FUNCTION_BLOCK FB_FieldCodecEnum EXTENDS FB_FieldCodec
VAR_INPUT
END_VAR
VAR_OUTPUT
END_VAR
VAR
	nValue : DINT;
END_VAR

METHOD CalculatePackedDataSize : HRESULT
VAR_INPUT CONSTANT
	anyFirstElem	: T_Any;
	nLength	        : UDINT;        // items to write
END_VAR
VAR_OUTPUT
    nPackedDataSize : UDINT;
END_VAR
VAR
    anyItem         : T_ANY;
    i               : UDINT;
END_VAR
IF anyFirstElem.pValue = NULL OR anyFirstElem.TypeClass <> __SYSTEM.TYPE_CLASS.TYPE_ENUM THEN
    CalculatePackedDataSize := E_HRESULTAdsErr.INVALIDDATA;
    RETURN;
END_IF

anyItem := anyFirstElem;

IF nLength < 1 THEN
    nPackedDataSize := 0;
    RETURN;
END_IF

FOR i := 0  TO nLength - 1 DO
    anyItem.pValue := anyFirstElem.pValue + (i * TO_UDINT(anyFirstElem.diSize)); 
    nPackedDataSize := nPackedDataSize + F_ComputeEnumSize(anyItem);
END_FOR
END_METHOD

METHOD IsPackedRepeatedField : BOOL
VAR_INPUT
	nTag	: UDINT;
END_VAR
IsPackedRepeatedField := F_IsPackedRepeatedField(nTag);
END_METHOD


METHOD ValueReader : HRESULT
VAR_IN_OUT      
    stCtx : ST_ParseContext;
END_VAR
VAR_OUTPUT
	anyOut	: T_Any;
END_VAR

ValueReader := F_ParseRawVarint32(stCtx, nValue);
IF FAILED(ValueReader) THEN
    RETURN;
END_IF
anyOut := F_ToAnyType(anyArg:= nValue);
END_METHOD

METHOD ValueWriter : HRESULT
VAR_IN_OUT
    stCtx  : ST_WriteContext;
END_VAR
VAR_INPUT
    anyIn : T_ANY;
END_VAR
VAR
    nValue  : DINT;
END_VAR
IF anyIn.pValue = NULL OR anyIn.TypeClass <> __SYSTEM.TYPE_CLASS.TYPE_ENUM THEN
    ValueWriter := E_HRESULTAdsErr.INVALIDDATA;
    RETURN;
END_IF

MEMCPY(destAddr:= ADR(nValue), srcAddr:= anyIn.pValue, MIN(TO_UDINT(anyIn.diSize), SIZEOF(nValue)));
ValueWriter := F_WriteInt32(stCtx, nValue);
END_METHOD

END_FUNCTION_BLOCK

(* stored: Version 1.1.0.1
   POU FB_FieldCodecEnum: Id {51053c22-4fc8-47e3-930a-74eb4c9c8e6a}, SpecialFunc None
   Method CalculatePackedDataSize: Id {cd558771-2c71-46d8-87c3-13f30229ace5}
   Method IsPackedRepeatedField: Id {3fa064e7-89fe-46ba-96c5-ce2eb0fee077}
   Method ValueReader: Id {96a03a26-650a-464a-9307-8361516bd3b2}
   Method ValueWriter: Id {fd6adb85-9839-4b56-95d2-db99fcdba5be} *)
